(* PLC project v0.6.02_RefactorGateAndTest.project, CODESYS CODESYS V3.5 SP19 Patch 1 *)
(* stored: creationDateTime 2026-08-15T23:16:29.358315, modificationDateTime 2026-08-15T23:16:29.358315 *)

(* ═══════════════════════════════════════════════════════════════ 💾 FB_SnapshotExporter — Moteur fichier CSV commun (CAA File) ─────────────────────────────────────────────────────────────── 🎯 Rôle : écrit un snapshot CSV sur front de bit, machine d'état multi-scan (IDLE→OPEN→WRITE→CLOSE→DONE/ERROR), 1 chunk/scan. 🔒 Polarité : TRUE = action/état actif ; FALSE = repos. 🧩 Architecture : FB technique non-mouvement, lecture seule + fichier. 📄 Docs : DOC/AF/AF_Partie-12_Fonction_Diagnostic/FB_SnapshotTroubleshooting_v1.0.md · DOC/AF/AF_Partie-12_Fonction_Diagnostic/FB_SnapshotIHM_v1.0.md ═══════════════════════════════════════════════════════════════ *)
TYPE ST_SnapshotColumn : STRUCT
  Name : STRING(80);  (* Nom de la colonne (condensé) *)
  Value : STRING(80);  (* Valeur convertie en texte *)
END_STRUCT;
END_TYPE
